(*^^^^^^^^^^^^^^^^^^^^^^^^^^^^^^^^^^^^^^ General Visualization ^^^^^^^^^^^^^^^^^^^^^^^^^^^^^^^^^^^^*)
	(*For Ready to Load Indicators*)
		(*Flash when tool should be loaded but load is not complete*)
		IF In_Auto AND Tool_At_Home AND NOT Welding_Complete AND All_Robots_Clear AND NOT All_Sensors_On.2
			THEN
				Ready_To_Load:= Pulse_500mS;
				(*Go solid when tool has been loaded properly*)
				(*Go solid when tool is ready to be unloaded*)
		ELSIF In_Auto AND All_Robots_Clear  AND ((Tool_At_Home AND NOT Welding_Complete AND All_Sensors_On.2 AND NOT Enable_Motion)
			OR (Tool_At_Unload.0 AND Welding_Complete AND (Sealing_Complete OR Sealer_Bypass) AND (Stud_Complete OR Stud_Bypass) AND TurntableA_At_Robot AND NOT All_Sensors_Off))
			THEN
				Ready_To_Load:= TRUE;
		ELSE
				Ready_To_Load:= FALSE;
		END_IF;
	(*For Red Stack Light Indicators*)
		Red_Lamp_Req:= PPFaults<>0 OR CLFaulted.0 OR CLFaulted.4 OR (NOT Sealer_Bypass AND MAIN.SL01.Disp1_Volume_NotOK AND (MAIN.R1.Task_ID_Ack=Seal_Fix16)) OR Load_Seq01.Faulted;


	(*Status Banners*)
		(*1 - Check Parts On Sub Check*)
		IF In_Auto AND NOT In_Manual AND NOT Cycle_Complete AND Tool_At_Load.0
			AND NOT Start_Load_Robots1 AND NOT Start_Load_Robots2 AND NOT Start_Seal_Robots AND NOT Start_Stud_Robots AND NOT Start_TurntableA
			AND NOT Start_TurntableB AND NOT Start_Weld_Robots AND NOT Start_Unload_Robots1 AND NOT Start_Unload_Robots2
			THEN
				IF NOT Dry_Cycle AND NOT All_Sensors_On.0
					THEN Status:= 1;
				ELSIF Dry_Cycle AND NOT Load_Complete1
					THEN Status:=1;
				END_IF;
		END_IF;
		(*2 - Sub Check OK*)
		IF In_Auto AND NOT In_Manual AND NOT Cycle_Complete AND Tool_At_Load.1
			AND NOT Start_Load_Robots1 AND NOT Start_Load_Robots2 AND NOT Start_Seal_Robots AND NOT Start_Stud_Robots AND NOT Start_TurntableA
			AND NOT Start_TurntableB AND NOT Start_Weld_Robots AND NOT Start_Unload_Robots1 AND NOT Start_Unload_Robots2
			THEN
				IF NOT Dry_Cycle AND NOT All_Sensors_On.1
					THEN Status:= 2;
				ELSIF Dry_Cycle AND NOT Load_Complete2
					THEN Status:=2;
				END_IF;
		END_IF;
		(*3 - Load Main Part*)
		IF In_Auto AND NOT In_Manual AND NOT Cycle_Complete AND Tool_At_Home
			AND NOT Start_Load_Robots1 AND NOT Start_Load_Robots2 AND NOT Start_Seal_Robots AND NOT Start_Stud_Robots AND NOT Start_TurntableA
			AND NOT Start_TurntableB AND NOT Start_Weld_Robots AND NOT Start_Unload_Robots1 AND NOT Start_Unload_Robots2
			THEN
				IF NOT Dry_Cycle AND NOT All_Sensors_On.2
					THEN Status:= 3;
				ELSIF Dry_Cycle AND NOT Load_Complete
					THEN Status:=3;
				END_IF;
		END_IF;
		(*10 - Load Parts Onto Tool*)
		IF In_Auto AND NOT In_Manual AND NOT Cycle_Complete AND Tool_At_Load.0
			AND NOT Start_Load_Robots1 AND NOT Start_Load_Robots2 AND NOT Start_Seal_Robots AND NOT Start_Stud_Robots AND NOT Start_TurntableA
			AND NOT Start_TurntableB AND NOT Start_Weld_Robots AND NOT Start_Unload_Robots1 AND NOT Start_Unload_Robots2
			THEN
				IF NOT Dry_Cycle AND NOT All_Sensors_On.2
					THEN Status:= 10;
				ELSIF Dry_Cycle AND NOT Load_Complete
					THEN Status:=10;
				END_IF;
		END_IF;
		(*11 - Robot(s) Loading*)
		IF ((Start_Load_Robots1 OR  Load_Robots_WorkingOK1) OR (Start_Load_Robots2 OR  Load_Robots_WorkingOK2)) AND In_Auto AND NOT In_Manual
			AND NOT Start_Seal_Robots AND NOT Start_Stud_Robots AND NOT Start_TurntableA
			AND NOT Start_TurntableB AND NOT Start_Weld_Robots AND NOT Start_Unload_Robots1 AND NOT Start_Unload_Robots2
			THEN Status:= 11;
		END_IF;
		(*12 - Parts Loaded OK*)
		IF In_Auto AND NOT In_Manual AND NOT Cycle_Complete
			AND NOT Start_Load_Robots1 AND NOT Start_Load_Robots2 AND NOT Start_Seal_Robots AND NOT Start_Stud_Robots AND NOT Start_TurntableA
			 AND NOT Start_TurntableB AND NOT Start_Weld_Robots AND NOT Start_Unload_Robots1 AND NOT Start_Unload_Robots2
			THEN
				IF (All_Sensors_On.2 AND Tool_At_Load.0) AND NOT Dry_Cycle
					THEN Status:= 12;
				ELSIF Load_Complete
					THEN Status:= 12;
				END_IF;
		END_IF;
		(*19 - Robot(s) Stud*)
		IF (Start_Stud_Robots OR Stud_Robots_WorkingOK) AND In_Auto AND NOT In_Manual
			AND NOT Start_Load_Robots1 AND NOT Start_Load_Robots2 AND NOT Start_Weld_Robots AND NOT Start_Seal_Robots AND NOT Start_TurntableA
			 AND NOT Start_TurntableB AND NOT Start_Unload_Robots1 AND NOT Start_Unload_Robots2
			THEN Status:= 19;
		END_IF;
		(*20 - Robot(s) Sealing*)
		IF (Start_Seal_Robots OR Seal_Robots_WorkingOK) AND In_Auto AND NOT In_Manual
			AND NOT Start_Load_Robots1 AND NOT Start_Load_Robots2 AND NOT Start_Weld_Robots AND NOT Start_Stud_Robots AND NOT Start_TurntableA
			 AND NOT Start_TurntableB AND NOT Start_Unload_Robots1 AND NOT Start_Unload_Robots2
			THEN Status:= 20;
		END_IF;
		(*21 - Robot(s) Welding*)
		IF (Start_Weld_Robots OR Weld_Robots_WorkingOK) AND In_Auto AND NOT In_Manual
			AND NOT Start_Load_Robots1 AND NOT Start_Load_Robots2 AND NOT Start_Seal_Robots AND NOT Start_Stud_Robots AND NOT Start_TurntableA
			 AND NOT Start_TurntableB AND NOT Start_Unload_Robots1 AND NOT Start_Unload_Robots2
			THEN Status:= 21;
		END_IF;
		(*22 - Welding Complete / Ready for Unload*)
		IF In_Auto AND NOT In_Manual AND NOT Cycle_Complete AND Welding_Complete
			AND NOT Start_Load_Robots1 AND NOT Start_Load_Robots2 AND NOT Start_Seal_Robots AND NOT Start_Stud_Robots AND NOT Start_TurntableA
			AND NOT Start_TurntableB AND NOT Start_Weld_Robots AND NOT Start_Unload_Robots1 AND NOT Start_Unload_Robots2
			THEN Status:= 22;
		END_IF;
		(*26 - Ready for Rotate*)
		IF (Start_TurntableA OR Start_TurntableB) AND In_Auto AND NOT In_Manual
			AND NOT Start_Load_Robots1 AND NOT Start_Load_Robots2 AND NOT Start_Seal_Robots AND NOT Start_Stud_Robots
			AND NOT Start_Weld_Robots AND NOT Start_Unload_Robots1 AND NOT Start_Unload_Robots2
			THEN Status := 26;
		END_IF;
		(*31 - Robot(s) Unloading*)
		IF (Start_Unload_Robots1 OR Unload_Robots_WorkingOK1 OR Start_Unload_Robots2 OR Unload_Robots_WorkingOK2) AND In_Auto AND NOT In_Manual
			AND NOT Start_Load_Robots1 AND NOT Start_Load_Robots2 AND NOT Start_Seal_Robots AND NOT Start_Stud_Robots AND NOT Start_TurntableA
			AND NOT Start_TurntableB AND NOT Start_Weld_Robots
			THEN Status:= 31;
		END_IF;
		(*32 - Unload Complete*)
		IF In_Auto AND NOT In_Manual AND NOT Cycle_Complete AND Unload_Complete
			AND NOT Start_Load_Robots1 AND NOT Start_Load_Robots2 AND NOT Start_Seal_Robots AND NOT Start_Stud_Robots AND NOT Start_TurntableA
			AND NOT Start_TurntableB AND NOT Start_Weld_Robots AND NOT Start_Unload_Robots1 AND NOT Start_Unload_Robots2
			THEN Status:= 32;
		END_IF;
		(*42 - Cycle Complete*)
		IF In_Auto AND NOT In_Manual AND Cycle_Complete AND All_Sensors_Off
			THEN Status:= 42;
		END_IF;
		(*50 - In Manual*)
		IF In_Manual
			THEN Status:= 50;
		END_IF;
		(*51 - Clamp Fault*)
		IF (CLFaults1>0 OR CLFaults2>0 OR CLFaults3>0 OR CLFaults4>0) AND In_Auto AND NOT In_Manual
			THEN Status:= 51;
		END_IF;
		(*52 - Part Present Sensor Fault*)
		IF PPFaults>0 AND In_Auto AND NOT In_Manual
			THEN Status:= 52;
		END_IF;
		(*53 - Nut Checks Failed Call QA*)
		IF QAChecks_Failed AND In_Auto AND NOT In_Manual
			THEN Status:= 53;
		END_IF;
		(*54 - Sealer Failed Call QA*)
		IF NOT Sealer_Bypass AND (MAIN.SL01.Disp1_Volume_NotOK AND (MAIN.R1.Task_ID_Ack=Seal_Fix16)) AND In_Auto AND NOT In_Manual
			THEN Status:= 54;
		END_IF;
		(*55 - Load Sequence Fault Call QA*)
		IF Load_Seq01.Faulted AND In_Auto AND NOT In_Manual
			THEN Status:= 55;
		END_IF;



(*$$$$$$$$$$$$$$$$$$$$$$$$$$$$$$$$$$$$$$$$$$$$$$$$$$$ Faults $$$$$$$$$$$$$$$$$$$$$$$$$$$$$$$$$$$$$$$$$$$$$$$$$$$$$$$*)

	(*Clamp/Cylider Faults Group 1*)
		IF CLFaults1>0
			THEN CLFaulted.1:=TRUE;
		ELSE
			CLFaulted.1:=FALSE;
		END_IF;
	(*Clamp/Cylider Faults Group 2*)
		IF CLFaults2>0
			THEN CLFaulted.2:=TRUE;
		ELSE
			CLFaulted.2:=FALSE;
		END_IF;
	(*Clamp/Cylider Faults Group 3*)
		IF CLFaults3>0
			THEN CLFaulted.3:=TRUE;
		ELSE
			CLFaulted.3:=FALSE;
		END_IF;
	(*Clamp/Cylinder Faults Group 4 - Reserved Flag for QA Check Motion Faults*)
		IF CLFaults4>0
			THEN CLFaulted.4:=TRUE;
		ELSE
			CLFaulted.4:=FALSE;
		END_IF;
	(*Bit 0 is designated as ANY Clamp Group Faulted*)
	IF CLFaulted.1 OR CLFaulted.2 OR CLFaulted.3
		THEN CLFaulted.0:= TRUE;
	ELSE CLFaulted.0 := FALSE;
	END_IF;

	(*Part Present Sensor Faults*)
		IF (PPFaults>0) OR (PPFaults1>0) OR (PPFaults2>0)
			THEN PPFaulted.0:=TRUE;
		ELSE
			PPFaulted.0:=FALSE;
		END_IF;
























(*end*)
END_ACTION

ACTION Task_Fix_Model_IDs:


	(*Develop Task IDs - See Global Variable, "TaskID_Record"*)

	IF (Start_Load_Robots1 OR Start_Load_Robots2) AND Enable_Motion
		THEN Task_ID:= Dropoff_Fix112;
	ELSIF Start_Seal_Robots AND Enable_Motion
		THEN Task_ID:= Seal_Fix112;
	ELSIF Start_Stud_Robots AND Enable_Motion
		THEN Task_ID:= Stud_Fix112;
	ELSIF Start_Weld_Robots AND Enable_Motion
		THEN Task_ID:= Weld_Fix112;
	ELSIF Start_TurnTableA AND Enable_Motion
		THEN Task_ID:= Sweep_Fix112;
	ELSIF (Start_Unload_Robots1 OR Start_Unload_Robots2) AND Enable_Motion
		THEN Task_ID:= Pickup_Fix112;
	ELSE Task_ID:= 0;
	END_IF;

	(*Develop Fixture ID*)
	Fix_ID:= N00.ID;					(*In Future Map Beckhoff Dip Switch Data From IP67 Block to Here*)

	(*Develop Model ID*)
	Model_ID:= Discrete_In.ModelData;
END_ACTION

ACTION Tool_States:


(*+++++++++++THIS AREA IS CUSTOM PER INSTALLATION AND WILL HAVE TO BE MODIFIED PER +++++++++++++*)
(*+++++++++++THIS AREA IS CUSTOM PER INSTALLATION AND WILL HAVE TO BE MODIFIED PER +++++++++++++*)

	Tool_At_HOME:= Clamp1RETD AND Clamp2RETD AND Clamp3RETD AND Clamp4RETD
				AND Clamp5RETD AND Clamp6RETD AND Clamp7RETD AND Clamp8RETD
				AND Clamp9RETD AND Clamp10RETD AND Clamp11RETD AND Clamp12RETD
				AND Clamp13RETD AND Clamp14RETD AND Clamp15RETD AND Clamp16RETD
				AND Clamp17RETD AND Clamp18RETD AND Clamp19RETD AND Clamp20RETD
				AND Clamp21RETD AND Clamp22RETD AND Clamp23RETD AND Clamp24RETD
				AND Pin1ADVD AND Pin2ADVD AND Pin3ADVD AND Pin4ADVD AND Pin5ADVD AND Pin6ADVD AND Pin7ADVD
				AND Pin8ADVD AND Pin9ADVD AND Pin10ADVD AND Pin11ADVD AND Pin12ADVD AND Pin13ADVD AND Pin14ADVD
				AND Slide1RETD AND Slide2RETD AND Slide3RETD AND Slide4RETD AND Slide5RETD AND Slide6RETD
				AND Swing1ADVD AND Swing2ADVD AND Swing3ADVD AND Swing4ADVD AND Swing5ADVD AND Swing6ADVD;


	Tool_At_Load.0:=Clamp1RETD AND Clamp2RETD AND Clamp3RETD AND Clamp4RETD
				AND Clamp5RETD AND Clamp6RETD AND Clamp7RETD AND Clamp8RETD
				AND Clamp9RETD AND Clamp10RETD AND Clamp11RETD AND Clamp12RETD
				AND Clamp13RETD AND Clamp14RETD AND Clamp15RETD AND Clamp16RETD
				AND Clamp17RETD AND Clamp18RETD AND Clamp19RETD AND Clamp20RETD
				AND Clamp21RETD AND Clamp22RETD AND Clamp23RETD AND Clamp24RETD
				AND Pin1ADVD AND Pin2ADVD AND Pin3ADVD AND Pin4ADVD AND Pin5ADVD AND Pin6ADVD AND Pin7ADVD
				AND Pin8ADVD AND Pin9ADVD AND Pin10ADVD AND Pin11ADVD AND Pin12ADVD AND Pin13ADVD AND Pin14ADVD
				AND Slide1RETD AND Slide2RETD AND Slide3RETD AND Slide4RETD AND Slide5RETD AND Slide6RETD
				AND Swing1ADVD AND Swing2ADVD AND Swing3ADVD AND Swing4ADVD AND Swing5ADVD AND Swing6ADVD;
	Tool_At_Load.1:=FALSE;
	Tool_At_Load.2:= FALSE;
	Tool_At_Load.3:= FALSE;
	Tool_At_Load.4:= FALSE;


	Tool_At_Seal.0:= Clamp1ADVD AND Clamp2ADVD AND Clamp3ADVD AND Clamp4ADVD
				AND Clamp5ADVD AND Clamp6ADVD AND Clamp7ADVD AND Clamp8ADVD
				AND Clamp9ADVD AND Clamp10ADVD AND Clamp11ADVD AND Clamp12ADVD
				AND Clamp13ADVD AND Clamp14ADVD AND Clamp15ADVD AND Clamp16ADVD
				AND Clamp17ADVD AND Clamp18ADVD AND Clamp19ADVD AND Clamp20ADVD
				AND Clamp21ADVD AND Clamp22ADVD AND Clamp23ADVD AND Clamp24ADVD
				AND Pin1ADVD AND Pin2ADVD AND Pin3ADVD AND Pin4ADVD AND Pin5ADVD AND Pin6ADVD AND Pin7ADVD
				AND Pin8ADVD AND Pin9ADVD AND Pin10ADVD AND Pin11ADVD AND Pin12ADVD AND Pin13ADVD AND Pin14ADVD
				AND Slide1RETD AND Slide2RETD AND Slide3RETD AND Slide4RETD AND Slide5RETD AND Slide6RETD
				AND Swing1ADVD AND Swing2ADVD AND Swing3ADVD AND Swing4ADVD AND Swing5ADVD AND Swing6ADVD;
	Tool_At_Seal.1:= FALSE;
	Tool_At_Seal.2:= FALSE;
	Tool_At_Seal.3:= FALSE;
	Tool_At_Seal.4:= FALSE;


	Tool_At_Stud.0:= Clamp1ADVD AND Clamp2ADVD AND Clamp3ADVD AND Clamp4ADVD
				AND Clamp5ADVD AND Clamp6ADVD AND Clamp7ADVD AND Clamp8ADVD
				AND Clamp9ADVD AND Clamp10ADVD AND Clamp11ADVD AND Clamp12ADVD
				AND Clamp13ADVD AND Clamp14ADVD AND Clamp15ADVD AND Clamp16ADVD
				AND Clamp17ADVD AND Clamp18ADVD AND Clamp19ADVD AND Clamp20ADVD
				AND Clamp21ADVD AND Clamp22ADVD AND Clamp23ADVD AND Clamp24ADVD
				AND Pin1ADVD AND Pin2ADVD AND Pin3ADVD AND Pin4ADVD AND Pin5ADVD AND Pin6ADVD AND Pin7ADVD
				AND Pin8ADVD AND Pin9ADVD AND Pin10ADVD AND Pin11ADVD AND Pin12ADVD AND Pin13ADVD AND Pin14ADVD
				AND Slide1RETD AND Slide2RETD AND Slide3RETD AND Slide4RETD AND Slide5RETD AND Slide6RETD
				AND Swing1ADVD AND Swing2ADVD AND Swing3ADVD AND Swing4ADVD AND Swing5ADVD AND Swing6ADVD;
	Tool_At_Stud.1:= FALSE;
	Tool_At_Stud.2:= FALSE;
	Tool_At_Stud.3:= FALSE;
	Tool_At_Stud.4:= FALSE;


	Tool_At_Rotate.0:= Clamp1ADVD AND Clamp2ADVD AND Clamp3ADVD AND Clamp4ADVD
				AND Clamp5ADVD AND Clamp6ADVD AND Clamp7ADVD AND Clamp8ADVD
				AND Clamp9ADVD AND Clamp10ADVD AND Clamp11ADVD AND Clamp12ADVD
				AND Clamp13ADVD AND Clamp14ADVD AND Clamp15ADVD AND Clamp16ADVD
				AND Clamp17ADVD AND Clamp18ADVD AND Clamp19ADVD AND Clamp20ADVD
				AND Clamp21ADVD AND Clamp22ADVD AND Clamp23ADVD AND Clamp24ADVD
				AND Pin1ADVD AND Pin2ADVD AND Pin3ADVD AND Pin4ADVD AND Pin5ADVD AND Pin6ADVD AND Pin7ADVD
				AND Pin8ADVD AND Pin9ADVD AND Pin10ADVD AND Pin11ADVD AND Pin12ADVD AND Pin13ADVD AND Pin14ADVD
				AND Slide1RETD AND Slide2RETD AND Slide3RETD AND Slide4RETD AND Slide5RETD AND Slide6RETD
				AND Swing1ADVD AND Swing2ADVD AND Swing3ADVD AND Swing4ADVD AND Swing5ADVD AND Swing6ADVD;
	Tool_At_Rotate.1:= FALSE;
	Tool_At_Rotate.2:= FALSE;
	Tool_At_Rotate.3:= FALSE;
	Tool_At_Rotate.4:= FALSE;


	Tool_At_Weld.0:= Clamp1ADVD AND Clamp2ADVD AND Clamp3ADVD AND Clamp4ADVD
				AND Clamp5ADVD AND Clamp6ADVD AND Clamp7ADVD AND Clamp8ADVD
				AND Clamp9ADVD AND Clamp10ADVD AND Clamp11ADVD AND Clamp12ADVD
				AND Clamp13ADVD AND Clamp14ADVD AND Clamp15ADVD AND Clamp16ADVD
				AND Clamp17ADVD AND Clamp18ADVD AND Clamp19ADVD AND Clamp20ADVD
				AND Clamp21ADVD AND Clamp22ADVD AND Clamp23ADVD AND Clamp24ADVD
				AND Pin1ADVD AND Pin2ADVD AND Pin3ADVD AND Pin4ADVD AND Pin5ADVD AND Pin6ADVD AND Pin7ADVD
				AND Pin8ADVD AND Pin9ADVD AND Pin10ADVD AND Pin11ADVD AND Pin12ADVD AND Pin13ADVD AND Pin14ADVD
				AND Slide1RETD AND Slide2RETD AND Slide3RETD AND Slide4RETD AND Slide5RETD AND Slide6RETD
				AND Swing1ADVD AND Swing2ADVD AND Swing3ADVD AND Swing4ADVD AND Swing5ADVD AND Swing6ADVD;
	Tool_At_Weld.1:= FALSE;
	Tool_At_Weld.2:= FALSE;
	Tool_At_Weld.3:= FALSE;
	Tool_At_Weld.4:= FALSE;


	Tool_At_Unload.0:=Clamp1RETD AND Clamp2RETD AND Clamp3RETD AND Clamp4RETD
				AND Clamp5RETD AND Clamp6RETD AND Clamp7RETD AND Clamp8RETD
				AND Clamp9RETD AND Clamp10RETD AND Clamp11RETD AND Clamp12RETD
				AND Clamp13RETD AND Clamp14RETD AND Clamp15RETD AND Clamp16RETD
				AND Clamp17RETD AND Clamp18RETD AND Clamp19RETD AND Clamp20RETD
				AND Clamp21RETD AND Clamp22RETD AND Clamp23RETD AND Clamp24RETD
				AND Pin1RETD AND Pin2RETD AND Pin3RETD AND Pin4RETD AND Pin5RETD AND Pin6RETD AND Pin7RETD
				AND Pin8RETD AND Pin9RETD AND Pin10RETD AND Pin11RETD AND Pin12RETD AND Pin13RETD AND Pin14RETD
				AND Slide1ADVD AND Slide2ADVD AND Slide3ADVD AND Slide4ADVD AND Slide5ADVD AND Slide6ADVD
				AND Swing1RETD AND Swing2RETD AND Swing3RETD AND Swing4RETD AND Swing5RETD AND Swing6RETD;
	Tool_At_Unload.1:=FALSE;
	Tool_At_Unload.2:= FALSE;
	Tool_At_Unload.3:= FALSE;
	Tool_At_Unload.4:= FALSE;







































(*end*)
END_ACTION

ACTION Tool_VBSeq_Repos:
(*+++++++++++THIS AREA IS CUSTOM PER INSTALLATION AND WILL HAVE TO BE MODIFIED PER +++++++++++++*)
(*+++++++++++THIS AREA IS CUSTOM PER INSTALLATION AND WILL HAVE TO BE MODIFIED PER +++++++++++++*)


(*!!!!!!!!!!!!!!!!!!!!!!!!!!!!!!!!!!!!!!!!!! Tool Motion Control !!!!!!!!!!!!!!!!!!!!!!!!!!!!!!!*)

(*----------------------------------------- Camp / Unclamp Steps -------------------------------*)

(*$$$$$$$$$$$$$$$$$$$$$$$$$$$$$$$$$$ Develop Clamp and Unclamp Interlocks $$$$$$$$$$$$$$$$$$$$$$*)
(* Note: This is one method to create valve bank commands for clamp and unclamp sequencing
you are welcome to use the direct method as well*)

	(*Start Clamp Sequence*)
	(*First Stage Clamping*)
	Clamp_Step.0:= Auto_Run AND NOT Welding_Complete AND FALSE;
	(*Second Stage Clamping*)
	Clamp_Step.1:=  Clamp_Step.0 AND FALSE;
	(*Third Stage Clamping*)
	Clamp_Step.2:= Clamp_Step.1 AND FALSE;
	(*Forth Stage Clamping*)
	Clamp_Step.3:= Clamp_Step.2 AND FALSE;


	(*Start Unlcamp Sequence*)
	(*First Stage Unclamping*)
	Unclamp_Step.0:= Welding_Complete AND FALSE;
	(*Second Stage Unclamping*)
	Unclamp_Step.1:= Unclamp_Step.0 AND FALSE;
	(*Third Stage Unclamping*)
	Unclamp_Step.2:= Unclamp_Step.1 AND FALSE;
	(*Fourth Stage Unclamping*)
	Unclamp_Step.3:= Unclamp_Step.2 AND FALSE;



(*------------------------------------------- Repositions --------------------------------------*)

	(*Reposition Request#1*)
	IF FALSE
		THEN
			Repo_Reqs.0:= TRUE;
	END_IF;

	(*Reposition Request#2*)
	IF FALSE
		THEN
			Repo_Reqs.1:= TRUE;
	END_IF;

	(*Reposition Request#3*)
	IF FALSE
		THEN
			Repo_Reqs.2:= TRUE;
	END_IF;

	(*Reposition Request#4*)
	IF FALSE
		THEN
			Repo_Reqs.3:= TRUE;
	END_IF;

	(*Reposition Request#5*)
	IF FALSE
		THEN
			Repo_Reqs.4:= TRUE;
	END_IF;

	(*Reposition Request#6*)
	IF FALSE
		THEN
			Repo_Reqs.5:= TRUE;
	END_IF;

	(*Reposition Request#7*)
	IF FALSE
		THEN
			Repo_Reqs.6:= TRUE;
	END_IF;

	(*Reposition Request#8*)
	IF FALSE
		THEN
			Repo_Reqs.7:= TRUE;
	END_IF;

	(*Reset All Reposition Acks At the End Of Cycle*)
	IF Cycle_Complete
		THEN
			Repo_Reqs:= 0;
	END_IF;

(*------------------------- Reposition Acks ---------------------*)
	Repo_Ack.0:= Repo_Reqs.0 AND FALSE;
	Repo_Ack.1:= Repo_Reqs.1 AND FALSE;
	Repo_Ack.2:= Repo_Reqs.2 AND FALSE;
	Repo_Ack.3:= Repo_Reqs.3 AND FALSE;
	Repo_Ack.4:= Repo_Reqs.4 AND FALSE;
	Repo_Ack.5:= Repo_Reqs.5 AND FALSE;
	Repo_Ack.6:= Repo_Reqs.6 AND FALSE;
	Repo_Ack.7:= Repo_Reqs.7 AND FALSE;
END_ACTION

ACTION ValveBank1:


(*+++++++++++THIS AREA IS CUSTOM PER INSTALLATION AND WILL HAVE TO BE MODIFIED PER +++++++++++++*)
(*+++++++++++THIS AREA IS CUSTOM PER INSTALLATION AND WILL HAVE TO BE MODIFIED PER +++++++++++++*)
(*+++++++++++THIS AREA IS CUSTOM PER INSTALLATION AND WILL HAVE TO BE MODIFIED PER +++++++++++++*)

(*+++++++++++VALVE BANK 1 +++++++++++++*)
(*+++++++++++VALVE BANK 1 +++++++++++++*)
(*+++++++++++VALVE BANK 1 +++++++++++++*)


	(*Valve 1, A+B*)
	(*spare*)
		Valve1FB
			(
			Enable_Motion:= Enable_Motion ,
			Enable_Latch:= TRUE,					(*Enabling Runs Valve as detent type (maintained solenoids*)
			Enable_SideA_PreCharge:= FALSE,		(*Enabling Turns Side A PreCharge Active, reset when Side B is energized in Auto*)
			Enable_SideB_PreCharge:= FALSE,		(*Enabling Turns Side B PreCharge Active, reset when Side A is energized in Auto*)
			PreCharge_Time:= T#0.1S,
			Enable_Auto_Commands:= In_Auto,
			Enable_Manual_Commands:= In_Manual AND All_Robots_Clear,
			In_Manual_SideA_Command:= Discrete_In.ManReqs.0,
			In_Manual_SideB_Command:= (Discrete_In.ManReqs.1 OR Discrete_In.Go_Home),
			SideA_Indicator:= (Clamp1ADVD AND Clamp2ADVD AND Clamp3ADVD AND Clamp4ADVD),
			SideB_Indicator:= (Clamp1RETD AND Clamp2RETD AND Clamp3RETD AND Clamp4RETD) OR Manual_Ind_HomePrompt,
			TurnOn_SideA_SOL=> N100.Q.0,
			TurnOn_SideB_SOL=> N100.Q.1,
			TurnOn_SideA_Indicator=> Manual_Indicators1.0,
			TurnOn_SideB_Indicator=> Manual_Indicators1.1
			 );
		Valve1FB.In_Auto_SideA_Command:= FALSE;
		Valve1FB.In_Auto_SideB_Command:= FALSE;


	(*Valve 2, A+B*)
	(*spare*)
		Valve2FB
			(
			Enable_Motion:= Enable_Motion ,
			Enable_Latch:= TRUE,					(*Enabling Runs Valve as detent type (maintained solenoids*)
			Enable_SideA_PreCharge:= FALSE,		(*Enabling Turns Side A PreCharge Active, reset when Side B is energized in Auto*)
			Enable_SideB_PreCharge:= FALSE,		(*Enabling Turns Side B PreCharge Active, reset when Side A is energized in Auto*)
			PreCharge_Time:= T#0.10S,
			Enable_Auto_Commands:= In_Auto,
			Enable_Manual_Commands:= In_Manual AND All_Robots_Clear,
			In_Manual_SideA_Command:= Discrete_In.ManReqs.2,
			In_Manual_SideB_Command:= Discrete_In.ManReqs.3,
			SideA_Indicator:= FALSE,
			SideB_Indicator:= FALSE,
			TurnOn_SideA_SOL=> N100.Q.2,
			TurnOn_SideB_SOL=> N100.Q.3,
			TurnOn_SideA_Indicator=> Manual_Indicators1.2,
			TurnOn_SideB_Indicator=> Manual_Indicators1.3
			 );
		Valve2FB.In_Auto_SideA_Command:= FALSE;
		Valve2FB.In_Auto_SideB_Command:= FALSE;


	(*Valve 3, A+B*)
	(*spare*)
		Valve3FB
			(
			Enable_Motion:= Enable_Motion ,
			Enable_Latch:= TRUE,					(*Enabling Runs Valve as detent type (maintained solenoids*)
			Enable_SideA_PreCharge:= FALSE,		(*Enabling Turns Side A PreCharge Active, reset when Side B is energized in Auto*)
			Enable_SideB_PreCharge:= FALSE,		(*Enabling Turns Side B PreCharge Active, reset when Side A is energized in Auto*)
			PreCharge_Time:= T#0.10S,
			Enable_Auto_Commands:= In_Auto,
			Enable_Manual_Commands:= In_Manual AND All_Robots_Clear,
			In_Manual_SideA_Command:= Discrete_In.ManReqs.4,
			In_Manual_SideB_Command:= Discrete_In.ManReqs.5,
			SideA_Indicator:= FALSE,
			SideB_Indicator:= FALSE,
			TurnOn_SideA_SOL=> N100.Q.4,
			TurnOn_SideB_SOL=> N100.Q.5,
			TurnOn_SideA_Indicator=> Manual_Indicators1.4,
			TurnOn_SideB_Indicator=> Manual_Indicators1.5
			 );
		Valve3FB.In_Auto_SideA_Command:= FALSE;
		Valve3FB.In_Auto_SideB_Command:= FALSE;


	(*Valve 4, A+B*)
	(*spare*)
		Valve4FB
			(
			Enable_Motion:= Enable_Motion ,
			Enable_Latch:= TRUE,					(*Enabling Runs Valve as detent type (maintained solenoids*)
			Enable_SideA_PreCharge:= FALSE,		(*Enabling Turns Side A PreCharge Active, reset when Side B is energized in Auto*)
			Enable_SideB_PreCharge:= FALSE,		(*Enabling Turns Side B PreCharge Active, reset when Side A is energized in Auto*)
			PreCharge_Time:= T#0.10S,
			Enable_Auto_Commands:= In_Auto,
			Enable_Manual_Commands:= In_Manual AND All_Robots_Clear,
			In_Manual_SideA_Command:= Discrete_In.ManReqs.6,
			In_Manual_SideB_Command:= Discrete_In.ManReqs.7,
			SideA_Indicator:= FALSE,
			SideB_Indicator:= FALSE,
			TurnOn_SideA_SOL=> N100.Q.6,
			TurnOn_SideB_SOL=> N100.Q.7,
			TurnOn_SideA_Indicator=> Manual_Indicators1.6,
			TurnOn_SideB_Indicator=> Manual_Indicators1.7
			 );
		Valve4FB.In_Auto_SideA_Command:= FALSE;
		Valve4FB.In_Auto_SideB_Command:= FALSE;


	(*Valve 5, A+B*)
	(*spare*)
		Valve5FB
			(
			Enable_Motion:= Enable_Motion ,
			Enable_Latch:= TRUE,					(*Enabling Runs Valve as detent type (maintained solenoids*)
			Enable_SideA_PreCharge:= FALSE,		(*Enabling Turns Side A PreCharge Active, reset when Side B is energized in Auto*)
			Enable_SideB_PreCharge:= FALSE,		(*Enabling Turns Side B PreCharge Active, reset when Side A is energized in Auto*)
			PreCharge_Time:= T#0.10S,
			Enable_Auto_Commands:= In_Auto,
			Enable_Manual_Commands:= In_Manual AND All_Robots_Clear,
			In_Manual_SideA_Command:= Discrete_In.ManReqs.8,
			In_Manual_SideB_Command:= Discrete_In.ManReqs.9,
			SideA_Indicator:= FALSE,
			SideB_Indicator:= FALSE,
			TurnOn_SideA_SOL=> N100.Q.8,
			TurnOn_SideB_SOL=> N100.Q.9,
			TurnOn_SideA_Indicator=> Manual_Indicators1.8,
			TurnOn_SideB_Indicator=> Manual_Indicators1.9
			 );
		Valve5FB.In_Auto_SideA_Command:= FALSE;
		Valve5FB.In_Auto_SideB_Command:= FALSE;


	(*Valve 6, A+B*)
	(*spare*)
		Valve6FB
			(
			Enable_Motion:= Enable_Motion ,
			Enable_Latch:= TRUE,					(*Enabling Runs Valve as detent type (maintained solenoids*)
			Enable_SideA_PreCharge:= FALSE,		(*Enabling Turns Side A PreCharge Active, reset when Side B is energized in Auto*)
			Enable_SideB_PreCharge:= FALSE,		(*Enabling Turns Side B PreCharge Active, reset when Side A is energized in Auto*)
			PreCharge_Time:= T#0.10S,
			Enable_Auto_Commands:= In_Auto,
			Enable_Manual_Commands:= In_Manual AND All_Robots_Clear,
			In_Manual_SideA_Command:= Discrete_In.ManReqs.10,
			In_Manual_SideB_Command:= Discrete_In.ManReqs.11,
			SideA_Indicator:= FALSE,
			SideB_Indicator:= FALSE,
			TurnOn_SideA_SOL=> N100.Q.10,
			TurnOn_SideB_SOL=> N100.Q.11,
			TurnOn_SideA_Indicator=> Manual_Indicators1.10,
			TurnOn_SideB_Indicator=> Manual_Indicators1.11
			 );
		Valve6FB.In_Auto_SideA_Command:= FALSE;
		Valve6FB.In_Auto_SideB_Command:= FALSE;


	(*Valve 7, A+B*)
	(*spare*)
		Valve7FB
			(
			Enable_Motion:= Enable_Motion ,
			Enable_Latch:= TRUE,					(*Enabling Runs Valve as detent type (maintained solenoids*)
			Enable_SideA_PreCharge:= FALSE,		(*Enabling Turns Side A PreCharge Active, reset when Side B is energized in Auto*)
			Enable_SideB_PreCharge:= FALSE,		(*Enabling Turns Side B PreCharge Active, reset when Side A is energized in Auto*)
			PreCharge_Time:= T#0.10S,
			Enable_Auto_Commands:= In_Auto,
			Enable_Manual_Commands:= In_Manual AND All_Robots_Clear,
			In_Manual_SideA_Command:= Discrete_In.ManReqs.12,
			In_Manual_SideB_Command:= Discrete_In.ManReqs.13,
			SideA_Indicator:= FALSE,
			SideB_Indicator:= FALSE,
			TurnOn_SideA_SOL=> N100.Q.12,
			TurnOn_SideB_SOL=> N100.Q.13,
			TurnOn_SideA_Indicator=> Manual_Indicators1.12,
			TurnOn_SideB_Indicator=> Manual_Indicators1.13
			 );
		Valve7FB.In_Auto_SideA_Command:= FALSE;
		Valve7FB.In_Auto_SideB_Command:= FALSE;


	(*Valve 8, A+B*)
	(*spare*)
		Valve8FB
			(
			Enable_Motion:= Enable_Motion ,
			Enable_Latch:= TRUE,					(*Enabling Runs Valve as detent type (maintained solenoids*)
			Enable_SideA_PreCharge:= FALSE,		(*Enabling Turns Side A PreCharge Active, reset when Side B is energized in Auto*)
			Enable_SideB_PreCharge:= FALSE,		(*Enabling Turns Side B PreCharge Active, reset when Side A is energized in Auto*)
			PreCharge_Time:= T#0.10S,
			Enable_Auto_Commands:= In_Auto,
			Enable_Manual_Commands:= In_Manual AND All_Robots_Clear,
			In_Manual_SideA_Command:= Discrete_In.ManReqs.14,
			In_Manual_SideB_Command:= Discrete_In.ManReqs.15,
			SideA_Indicator:= FALSE,
			SideB_Indicator:= FALSE,
			TurnOn_SideA_SOL=> N100.Q.14,
			TurnOn_SideB_SOL=> N100.Q.15,
			TurnOn_SideA_Indicator=> Manual_Indicators1.14,
			TurnOn_SideB_Indicator=> Manual_Indicators1.15
			 );
		Valve8FB.In_Auto_SideA_Command:= FALSE;
		Valve8FB.In_Auto_SideB_Command:= FALSE;


	(*Valve 9, A+B*)
	(*spare*)
		Valve9FB
			(
			Enable_Motion:= Enable_Motion ,
			Enable_Latch:= TRUE,					(*Enabling Runs Valve as detent type (maintained solenoids*)
			Enable_SideA_PreCharge:= FALSE,		(*Enabling Turns Side A PreCharge Active, reset when Side B is energized in Auto*)
			Enable_SideB_PreCharge:= FALSE,		(*Enabling Turns Side B PreCharge Active, reset when Side A is energized in Auto*)
			PreCharge_Time:= T#0.10S,
			Enable_Auto_Commands:= In_Auto,
			Enable_Manual_Commands:= In_Manual AND All_Robots_Clear,
			In_Manual_SideA_Command:= Discrete_In.ManReqs.16,
			In_Manual_SideB_Command:= Discrete_In.ManReqs.17,
			SideA_Indicator:= FALSE,
			SideB_Indicator:= FALSE,
			TurnOn_SideA_SOL=> N100.Q.16,
			TurnOn_SideB_SOL=> N100.Q.17,
			TurnOn_SideA_Indicator=> Manual_Indicators1.16,
			TurnOn_SideB_Indicator=> Manual_Indicators1.17
			 );
		Valve9FB.In_Auto_SideA_Command:= FALSE;
		Valve9FB.In_Auto_SideB_Command:= FALSE;


	(*Valve 10, A+B*)
	(*spare*)
		Valve10FB
			(
			Enable_Motion:= Enable_Motion ,
			Enable_Latch:= TRUE,					(*Enabling Runs Valve as detent type (maintained solenoids*)
			Enable_SideA_PreCharge:= FALSE,		(*Enabling Turns Side A PreCharge Active, reset when Side B is energized in Auto*)
			Enable_SideB_PreCharge:= FALSE,		(*Enabling Turns Side B PreCharge Active, reset when Side A is energized in Auto*)
			PreCharge_Time:= T#0.10S,
			Enable_Auto_Commands:= In_Auto,
			Enable_Manual_Commands:= In_Manual AND All_Robots_Clear,
			In_Manual_SideA_Command:= Discrete_In.ManReqs.18,
			In_Manual_SideB_Command:= Discrete_In.ManReqs.19,
			SideA_Indicator:= FALSE,
			SideB_Indicator:= FALSE,
			TurnOn_SideA_SOL=> N100.Q.18,
			TurnOn_SideB_SOL=> N100.Q.19,
			TurnOn_SideA_Indicator=> Manual_Indicators1.18,
			TurnOn_SideB_Indicator=> Manual_Indicators1.19
			 );
		Valve10FB.In_Auto_SideA_Command:= FALSE;
		Valve10FB.In_Auto_SideB_Command:= FALSE;


	(*Valve 11, A+B*)
	(*spare*)
		Valve11FB
			(
			Enable_Motion:= Enable_Motion ,
			Enable_Latch:= TRUE,					(*Enabling Runs Valve as detent type (maintained solenoids*)
			Enable_SideA_PreCharge:= FALSE,		(*Enabling Turns Side A PreCharge Active, reset when Side B is energized in Auto*)
			Enable_SideB_PreCharge:= FALSE,		(*Enabling Turns Side B PreCharge Active, reset when Side A is energized in Auto*)
			PreCharge_Time:= T#0.10S,
			Enable_Auto_Commands:= In_Auto,
			Enable_Manual_Commands:= In_Manual AND All_Robots_Clear,
			In_Manual_SideA_Command:= Discrete_In.ManReqs.20,
			In_Manual_SideB_Command:= Discrete_In.ManReqs.21,
			SideA_Indicator:= FALSE,
			SideB_Indicator:= FALSE,
			TurnOn_SideA_SOL=> N100.Q.20,
			TurnOn_SideB_SOL=> N100.Q.21,
			TurnOn_SideA_Indicator=> Manual_Indicators1.20,
			TurnOn_SideB_Indicator=> Manual_Indicators1.21
			 );
		Valve11FB.In_Auto_SideA_Command:= FALSE;
		Valve11FB.In_Auto_SideB_Command:= FALSE;


	(*Valve 12, A+B*)
	(*spare*)
		Valve12FB
			(
			Enable_Motion:= Enable_Motion ,
			Enable_Latch:= TRUE,					(*Enabling Runs Valve as detent type (maintained solenoids*)
			Enable_SideA_PreCharge:= FALSE,		(*Enabling Turns Side A PreCharge Active, reset when Side B is energized in Auto*)
			Enable_SideB_PreCharge:= FALSE,		(*Enabling Turns Side B PreCharge Active, reset when Side A is energized in Auto*)
			PreCharge_Time:= T#0.10S,
			Enable_Auto_Commands:= In_Auto,
			Enable_Manual_Commands:= In_Manual AND All_Robots_Clear,
			In_Manual_SideA_Command:= Discrete_In.ManReqs.22,
			In_Manual_SideB_Command:= Discrete_In.ManReqs.23,
			SideA_Indicator:= FALSE,
			SideB_Indicator:= FALSE,
			TurnOn_SideA_SOL=> N100.Q.22,
			TurnOn_SideB_SOL=> N100.Q.23,
			TurnOn_SideA_Indicator=> Manual_Indicators1.22,
			TurnOn_SideB_Indicator=> Manual_Indicators1.23
			 );
		Valve12FB.In_Auto_SideA_Command:= FALSE;
		Valve12FB.In_Auto_SideB_Command:= FALSE;


	(*Valve 13, A+B*)
	(*spare*)
		Valve13FB
			(
			Enable_Motion:= Enable_Motion ,
			Enable_Latch:= TRUE,					(*Enabling Runs Valve as detent type (maintained solenoids*)
			Enable_SideA_PreCharge:= FALSE,		(*Enabling Turns Side A PreCharge Active, reset when Side B is energized in Auto*)
			Enable_SideB_PreCharge:= FALSE,		(*Enabling Turns Side B PreCharge Active, reset when Side A is energized in Auto*)
			PreCharge_Time:= T#0.10S,
			Enable_Auto_Commands:= In_Auto,
			Enable_Manual_Commands:= In_Manual AND All_Robots_Clear,
			In_Manual_SideA_Command:= Discrete_In.ManReqs.24,
			In_Manual_SideB_Command:= Discrete_In.ManReqs.25,
			SideA_Indicator:= FALSE,
			SideB_Indicator:= FALSE,
			TurnOn_SideA_SOL=> N100.Q.24,
			TurnOn_SideB_SOL=> N100.Q.25,
			TurnOn_SideA_Indicator=> Manual_Indicators1.24,
			TurnOn_SideB_Indicator=> Manual_Indicators1.25
			 );
		Valve13FB.In_Auto_SideA_Command:= FALSE;
		Valve13FB.In_Auto_SideB_Command:= FALSE;


	(*Valve 14, A+B*)
	(*spare*)
		Valve14FB
			(
			Enable_Motion:= Enable_Motion ,
			Enable_Latch:= TRUE,					(*Enabling Runs Valve as detent type (maintained solenoids*)
			Enable_SideA_PreCharge:= FALSE,		(*Enabling Turns Side A PreCharge Active, reset when Side B is energized in Auto*)
			Enable_SideB_PreCharge:= FALSE,		(*Enabling Turns Side B PreCharge Active, reset when Side A is energized in Auto*)
			PreCharge_Time:= T#0.10S,
			Enable_Auto_Commands:= In_Auto,
			Enable_Manual_Commands:= In_Manual AND All_Robots_Clear,
			In_Manual_SideA_Command:= Discrete_In.ManReqs.26,
			In_Manual_SideB_Command:= Discrete_In.ManReqs.27,
			SideA_Indicator:= FALSE,
			SideB_Indicator:= FALSE,
			TurnOn_SideA_SOL=> N100.Q.26,
			TurnOn_SideB_SOL=> N100.Q.27,
			TurnOn_SideA_Indicator=> Manual_Indicators1.26,
			TurnOn_SideB_Indicator=> Manual_Indicators1.27
			 );
		Valve14FB.In_Auto_SideA_Command:= FALSE;
		Valve14FB.In_Auto_SideB_Command:= FALSE;


	(*Valve 15, A+B*)
	(*spare*)
		Valve15FB
			(
			Enable_Motion:= Enable_Motion ,
			Enable_Latch:= TRUE,					(*Enabling Runs Valve as detent type (maintained solenoids*)
			Enable_SideA_PreCharge:= FALSE,		(*Enabling Turns Side A PreCharge Active, reset when Side B is energized in Auto*)
			Enable_SideB_PreCharge:= FALSE,		(*Enabling Turns Side B PreCharge Active, reset when Side A is energized in Auto*)
			PreCharge_Time:= T#0.10S,
			Enable_Auto_Commands:= In_Auto,
			Enable_Manual_Commands:= In_Manual AND All_Robots_Clear,
			In_Manual_SideA_Command:= Discrete_In.ManReqs.28,
			In_Manual_SideB_Command:= Discrete_In.ManReqs.29,
			SideA_Indicator:= FALSE,
			SideB_Indicator:= FALSE,
			TurnOn_SideA_SOL=> N100.Q.28,
			TurnOn_SideB_SOL=> N100.Q.29,
			TurnOn_SideA_Indicator=> Manual_Indicators1.28,
			TurnOn_SideB_Indicator=> Manual_Indicators1.29
			 );
		Valve15FB.In_Auto_SideA_Command:= FALSE;
		Valve15FB.In_Auto_SideB_Command:= FALSE;


	(*Valve 16, A+B*)
	(*spare*)
		Valve16FB
			(
			Enable_Motion:= Enable_Motion ,
			Enable_Latch:= TRUE,					(*Enabling Runs Valve as detent type (maintained solenoids*)
			Enable_SideA_PreCharge:= FALSE,		(*Enabling Turns Side A PreCharge Active, reset when Side B is energized in Auto*)
			Enable_SideB_PreCharge:= FALSE,		(*Enabling Turns Side B PreCharge Active, reset when Side A is energized in Auto*)
			PreCharge_Time:= T#0.10S,
			Enable_Auto_Commands:= In_Auto,
			Enable_Manual_Commands:= In_Manual AND All_Robots_Clear,
			In_Manual_SideA_Command:= Discrete_In.ManReqs.30,
			In_Manual_SideB_Command:= Discrete_In.ManReqs.31,
			SideA_Indicator:= FALSE,
			SideB_Indicator:= FALSE,
			TurnOn_SideA_SOL=> N100.Q.30,
			TurnOn_SideB_SOL=> N100.Q.31,
			TurnOn_SideA_Indicator=> Manual_Indicators1.30,
			TurnOn_SideB_Indicator=> Manual_Indicators1.31
			 );
		Valve16FB.In_Auto_SideA_Command:= FALSE;
		Valve16FB.In_Auto_SideB_Command:= FALSE;


























(*end*)
END_ACTION

ACTION ValveBank2:


(*+++++++++++THIS AREA IS CUSTOM PER INSTALLATION AND WILL HAVE TO BE MODIFIED PER +++++++++++++*)
(*+++++++++++THIS AREA IS CUSTOM PER INSTALLATION AND WILL HAVE TO BE MODIFIED PER +++++++++++++*)
(*+++++++++++THIS AREA IS CUSTOM PER INSTALLATION AND WILL HAVE TO BE MODIFIED PER +++++++++++++*)

(*+++++++++++VALVE BANK 2 +++++++++++++*)
(*+++++++++++VALVE BANK 2 +++++++++++++*)
(*+++++++++++VALVE BANK 2 +++++++++++++*)


	(*Valve 17, A+B*)
	(*spare*)
		Valve17FB
			(
			Enable_Motion:= Enable_Motion ,
			Enable_Latch:= TRUE,					(*Enabling Runs Valve as detent type (maintained solenoids*)
			Enable_SideA_PreCharge:= FALSE,		(*Enabling Turns Side A PreCharge Active, reset when Side B is energized in Auto*)
			Enable_SideB_PreCharge:= FALSE,		(*Enabling Turns Side B PreCharge Active, reset when Side A is energized in Auto*)
			PreCharge_Time:= T#0.1S,
			Enable_Auto_Commands:= In_Auto,
			Enable_Manual_Commands:= In_Manual AND All_Robots_Clear,
			In_Manual_SideA_Command:= Discrete_In.ManReqs2.0,
			In_Manual_SideB_Command:= (Discrete_In.ManReqs2.1 OR Discrete_In.Go_Home),
			SideA_Indicator:= FALSE,
			SideB_Indicator:= FALSE,
			TurnOn_SideA_SOL=> N101.Q.0,
			TurnOn_SideB_SOL=> N101.Q.1,
			TurnOn_SideA_Indicator=> Manual_Indicators2.0,
			TurnOn_SideB_Indicator=> Manual_Indicators2.1
			 );
		Valve17FB.In_Auto_SideA_Command:= FALSE;
		Valve17FB.In_Auto_SideB_Command:= FALSE;


	(*Valve 18, A+B*)
	(*spare*)
		Valve18FB
			(
			Enable_Motion:= Enable_Motion ,
			Enable_Latch:= TRUE,					(*Enabling Runs Valve as detent type (maintained solenoids*)
			Enable_SideA_PreCharge:= FALSE,		(*Enabling Turns Side A PreCharge Active, reset when Side B is energized in Auto*)
			Enable_SideB_PreCharge:= FALSE,		(*Enabling Turns Side B PreCharge Active, reset when Side A is energized in Auto*)
			PreCharge_Time:= T#0.10S,
			Enable_Auto_Commands:= In_Auto,
			Enable_Manual_Commands:= In_Manual AND All_Robots_Clear,
			In_Manual_SideA_Command:= Discrete_In.ManReqs2.2,
			In_Manual_SideB_Command:= Discrete_In.ManReqs2.3,
			SideA_Indicator:= FALSE,
			SideB_Indicator:= FALSE,
			TurnOn_SideA_SOL=> N101.Q.2,
			TurnOn_SideB_SOL=> N101.Q.3,
			TurnOn_SideA_Indicator=> Manual_Indicators2.2,
			TurnOn_SideB_Indicator=> Manual_Indicators2.3
			 );
		Valve18FB.In_Auto_SideA_Command:= FALSE;
		Valve18FB.In_Auto_SideB_Command:= FALSE;

	(*Valve 19, A+B*)
	(*spare*)
		Valve19FB
			(
			Enable_Motion:= Enable_Motion ,
			Enable_Latch:= TRUE,					(*Enabling Runs Valve as detent type (maintained solenoids*)
			Enable_SideA_PreCharge:= FALSE,		(*Enabling Turns Side A PreCharge Active, reset when Side B is energized in Auto*)
			Enable_SideB_PreCharge:= FALSE,		(*Enabling Turns Side B PreCharge Active, reset when Side A is energized in Auto*)
			PreCharge_Time:= T#0.10S,
			Enable_Auto_Commands:= In_Auto,
			Enable_Manual_Commands:= In_Manual AND All_Robots_Clear,
			In_Manual_SideA_Command:= Discrete_In.ManReqs2.4,
			In_Manual_SideB_Command:= Discrete_In.ManReqs2.5,
			SideA_Indicator:= FALSE,
			SideB_Indicator:= FALSE,
			TurnOn_SideA_SOL=> N101.Q.4,
			TurnOn_SideB_SOL=> N101.Q.5,
			TurnOn_SideA_Indicator=> Manual_Indicators2.4,
			TurnOn_SideB_Indicator=> Manual_Indicators2.5
			 );
		Valve19FB.In_Auto_SideA_Command:= FALSE;
		Valve19FB.In_Auto_SideB_Command:= FALSE;


	(*Valve 20, A+B*)
	(*spare*)
		Valve20FB
			(
			Enable_Motion:= Enable_Motion ,
			Enable_Latch:= TRUE,					(*Enabling Runs Valve as detent type (maintained solenoids*)
			Enable_SideA_PreCharge:= FALSE,		(*Enabling Turns Side A PreCharge Active, reset when Side B is energized in Auto*)
			Enable_SideB_PreCharge:= FALSE,		(*Enabling Turns Side B PreCharge Active, reset when Side A is energized in Auto*)
			PreCharge_Time:= T#0.10S,
			Enable_Auto_Commands:= In_Auto,
			Enable_Manual_Commands:= In_Manual AND All_Robots_Clear,
			In_Manual_SideA_Command:= Discrete_In.ManReqs2.6,
			In_Manual_SideB_Command:= Discrete_In.ManReqs2.7,
			SideA_Indicator:= FALSE,
			SideB_Indicator:= FALSE,
			TurnOn_SideA_SOL=> N101.Q.6,
			TurnOn_SideB_SOL=> N101.Q.7,
			TurnOn_SideA_Indicator=> Manual_Indicators2.6,
			TurnOn_SideB_Indicator=> Manual_Indicators2.7
			 );
		Valve20FB.In_Auto_SideA_Command:= FALSE;
		Valve20FB.In_Auto_SideB_Command:= FALSE;


	(*Valve 21, A+B*)
	(*spare*)
		Valve21FB
			(
			Enable_Motion:= Enable_Motion ,
			Enable_Latch:= TRUE,					(*Enabling Runs Valve as detent type (maintained solenoids*)
			Enable_SideA_PreCharge:= FALSE,		(*Enabling Turns Side A PreCharge Active, reset when Side B is energized in Auto*)
			Enable_SideB_PreCharge:= FALSE,		(*Enabling Turns Side B PreCharge Active, reset when Side A is energized in Auto*)
			PreCharge_Time:= T#0.10S,
			Enable_Auto_Commands:= In_Auto,
			Enable_Manual_Commands:= In_Manual AND All_Robots_Clear,
			In_Manual_SideA_Command:= Discrete_In.ManReqs2.8,
			In_Manual_SideB_Command:= Discrete_In.ManReqs2.9,
			SideA_Indicator:= FALSE,
			SideB_Indicator:= FALSE,
			TurnOn_SideA_SOL=> N101.Q.8,
			TurnOn_SideB_SOL=> N101.Q.9,
			TurnOn_SideA_Indicator=> Manual_Indicators2.8,
			TurnOn_SideB_Indicator=> Manual_Indicators2.9
			 );
		Valve21FB.In_Auto_SideA_Command:= FALSE;
		Valve21FB.In_Auto_SideB_Command:= FALSE;


	(*Valve 22, A+B*)
	(*spare*)
		Valve22FB
			(
			Enable_Motion:= Enable_Motion ,
			Enable_Latch:= TRUE,					(*Enabling Runs Valve as detent type (maintained solenoids*)
			Enable_SideA_PreCharge:= FALSE,		(*Enabling Turns Side A PreCharge Active, reset when Side B is energized in Auto*)
			Enable_SideB_PreCharge:= FALSE,		(*Enabling Turns Side B PreCharge Active, reset when Side A is energized in Auto*)
			PreCharge_Time:= T#0.10S,
			Enable_Auto_Commands:= In_Auto,
			Enable_Manual_Commands:= In_Manual AND All_Robots_Clear,
			In_Manual_SideA_Command:= Discrete_In.ManReqs2.10,
			In_Manual_SideB_Command:= Discrete_In.ManReqs2.11,
			SideA_Indicator:= FALSE,
			SideB_Indicator:= FALSE,
			TurnOn_SideA_SOL=> N101.Q.10,
			TurnOn_SideB_SOL=> N101.Q.11,
			TurnOn_SideA_Indicator=> Manual_Indicators2.10,
			TurnOn_SideB_Indicator=> Manual_Indicators2.11
			 );
		Valve22FB.In_Auto_SideA_Command:= FALSE;
		Valve22FB.In_Auto_SideB_Command:= FALSE;


	(*Valve 23, A+B*)
	(*spare*)
		Valve23FB
			(
			Enable_Motion:= Enable_Motion ,
			Enable_Latch:= TRUE,					(*Enabling Runs Valve as detent type (maintained solenoids*)
			Enable_SideA_PreCharge:= FALSE,		(*Enabling Turns Side A PreCharge Active, reset when Side B is energized in Auto*)
			Enable_SideB_PreCharge:= FALSE,		(*Enabling Turns Side B PreCharge Active, reset when Side A is energized in Auto*)
			PreCharge_Time:= T#0.10S,
			Enable_Auto_Commands:= In_Auto,
			Enable_Manual_Commands:= In_Manual AND All_Robots_Clear,
			In_Manual_SideA_Command:= Discrete_In.ManReqs2.12,
			In_Manual_SideB_Command:= Discrete_In.ManReqs2.13,
			SideA_Indicator:= FALSE,
			SideB_Indicator:= FALSE,
			TurnOn_SideA_SOL=> N101.Q.12,
			TurnOn_SideB_SOL=> N101.Q.13,
			TurnOn_SideA_Indicator=> Manual_Indicators2.12,
			TurnOn_SideB_Indicator=> Manual_Indicators2.13
			 );
		Valve23FB.In_Auto_SideA_Command:= FALSE;
		Valve23FB.In_Auto_SideB_Command:= FALSE;


	(*Valve 24, A+B*)
	(*spare*)
		Valve24FB
			(
			Enable_Motion:= Enable_Motion ,
			Enable_Latch:= TRUE,					(*Enabling Runs Valve as detent type (maintained solenoids*)
			Enable_SideA_PreCharge:= FALSE,		(*Enabling Turns Side A PreCharge Active, reset when Side B is energized in Auto*)
			Enable_SideB_PreCharge:= FALSE,		(*Enabling Turns Side B PreCharge Active, reset when Side A is energized in Auto*)
			PreCharge_Time:= T#0.10S,
			Enable_Auto_Commands:= In_Auto,
			Enable_Manual_Commands:= In_Manual AND All_Robots_Clear,
			In_Manual_SideA_Command:= Discrete_In.ManReqs2.14,
			In_Manual_SideB_Command:= Discrete_In.ManReqs2.15,
			SideA_Indicator:= FALSE,
			SideB_Indicator:= FALSE,
			TurnOn_SideA_SOL=> N101.Q.14,
			TurnOn_SideB_SOL=> N101.Q.15,
			TurnOn_SideA_Indicator=> Manual_Indicators2.14,
			TurnOn_SideB_Indicator=> Manual_Indicators2.15
			 );
		Valve24FB.In_Auto_SideA_Command:= FALSE;
		Valve24FB.In_Auto_SideB_Command:= FALSE;


	(*Valve 25, A+B*)
	(*spare*)
		Valve25FB
			(
			Enable_Motion:= Enable_Motion ,
			Enable_Latch:= TRUE,					(*Enabling Runs Valve as detent type (maintained solenoids*)
			Enable_SideA_PreCharge:= FALSE,		(*Enabling Turns Side A PreCharge Active, reset when Side B is energized in Auto*)
			Enable_SideB_PreCharge:= FALSE,		(*Enabling Turns Side B PreCharge Active, reset when Side A is energized in Auto*)
			PreCharge_Time:= T#0.10S,
			Enable_Auto_Commands:= In_Auto,
			Enable_Manual_Commands:= In_Manual AND All_Robots_Clear,
			In_Manual_SideA_Command:= Discrete_In.ManReqs2.16,
			In_Manual_SideB_Command:= Discrete_In.ManReqs2.17,
			SideA_Indicator:= FALSE,
			SideB_Indicator:= FALSE,
			TurnOn_SideA_SOL=> N101.Q.16,
			TurnOn_SideB_SOL=> N101.Q.17,
			TurnOn_SideA_Indicator=> Manual_Indicators2.16,
			TurnOn_SideB_Indicator=> Manual_Indicators2.17
			 );
		Valve25FB.In_Auto_SideA_Command:= FALSE;
		Valve25FB.In_Auto_SideB_Command:= FALSE;


	(*Valve 26, A+B*)
	(*spare*)
		Valve26FB
			(
			Enable_Motion:= Enable_Motion ,
			Enable_Latch:= TRUE,					(*Enabling Runs Valve as detent type (maintained solenoids*)
			Enable_SideA_PreCharge:= FALSE,		(*Enabling Turns Side A PreCharge Active, reset when Side B is energized in Auto*)
			Enable_SideB_PreCharge:= FALSE,		(*Enabling Turns Side B PreCharge Active, reset when Side A is energized in Auto*)
			PreCharge_Time:= T#0.10S,
			Enable_Auto_Commands:= In_Auto,
			Enable_Manual_Commands:= In_Manual AND All_Robots_Clear,
			In_Manual_SideA_Command:= Discrete_In.ManReqs2.18,
			In_Manual_SideB_Command:= Discrete_In.ManReqs2.19,
			SideA_Indicator:= FALSE,
			SideB_Indicator:= FALSE,
			TurnOn_SideA_SOL=> N101.Q.18,
			TurnOn_SideB_SOL=> N101.Q.19,
			TurnOn_SideA_Indicator=> Manual_Indicators2.18,
			TurnOn_SideB_Indicator=> Manual_Indicators2.19
			 );
		Valve26FB.In_Auto_SideA_Command:= FALSE;
		Valve26FB.In_Auto_SideB_Command:= FALSE;


	(*Valve 27, A+B*)
	(*spare*)
		Valve27FB
			(
			Enable_Motion:= Enable_Motion ,
			Enable_Latch:= TRUE,					(*Enabling Runs Valve as detent type (maintained solenoids*)
			Enable_SideA_PreCharge:= FALSE,		(*Enabling Turns Side A PreCharge Active, reset when Side B is energized in Auto*)
			Enable_SideB_PreCharge:= FALSE,		(*Enabling Turns Side B PreCharge Active, reset when Side A is energized in Auto*)
			PreCharge_Time:= T#0.10S,
			Enable_Auto_Commands:= In_Auto,
			Enable_Manual_Commands:= In_Manual AND All_Robots_Clear,
			In_Manual_SideA_Command:= Discrete_In.ManReqs2.20,
			In_Manual_SideB_Command:= Discrete_In.ManReqs2.21,
			SideA_Indicator:= FALSE,
			SideB_Indicator:= FALSE,
			TurnOn_SideA_SOL=> N101.Q.20,
			TurnOn_SideB_SOL=> N101.Q.21,
			TurnOn_SideA_Indicator=> Manual_Indicators2.20,
			TurnOn_SideB_Indicator=> Manual_Indicators2.21
			 );
		Valve27FB.In_Auto_SideA_Command:= FALSE;
		Valve27FB.In_Auto_SideB_Command:= FALSE;


	(*Valve 28, A+B*)
	(*spare*)
		Valve28FB
			(
			Enable_Motion:= Enable_Motion ,
			Enable_Latch:= TRUE,					(*Enabling Runs Valve as detent type (maintained solenoids*)
			Enable_SideA_PreCharge:= FALSE,		(*Enabling Turns Side A PreCharge Active, reset when Side B is energized in Auto*)
			Enable_SideB_PreCharge:= FALSE,		(*Enabling Turns Side B PreCharge Active, reset when Side A is energized in Auto*)
			PreCharge_Time:= T#0.10S,
			Enable_Auto_Commands:= In_Auto,
			Enable_Manual_Commands:= In_Manual AND All_Robots_Clear,
			In_Manual_SideA_Command:= Discrete_In.ManReqs2.22,
			In_Manual_SideB_Command:= Discrete_In.ManReqs2.23,
			SideA_Indicator:= FALSE,
			SideB_Indicator:= FALSE,
			TurnOn_SideA_SOL=> N101.Q.22,
			TurnOn_SideB_SOL=> N101.Q.23,
			TurnOn_SideA_Indicator=> Manual_Indicators2.22,
			TurnOn_SideB_Indicator=> Manual_Indicators2.23
			 );
		Valve28FB.In_Auto_SideA_Command:= FALSE;
		Valve28FB.In_Auto_SideB_Command:= FALSE;


	(*Valve 29, A+B*)
	(*spare*)
		Valve29FB
			(
			Enable_Motion:= Enable_Motion ,
			Enable_Latch:= TRUE,					(*Enabling Runs Valve as detent type (maintained solenoids*)
			Enable_SideA_PreCharge:= FALSE,		(*Enabling Turns Side A PreCharge Active, reset when Side B is energized in Auto*)
			Enable_SideB_PreCharge:= FALSE,		(*Enabling Turns Side B PreCharge Active, reset when Side A is energized in Auto*)
			PreCharge_Time:= T#0.10S,
			Enable_Auto_Commands:= In_Auto,
			Enable_Manual_Commands:= In_Manual AND All_Robots_Clear,
			In_Manual_SideA_Command:= Discrete_In.ManReqs2.24,
			In_Manual_SideB_Command:= Discrete_In.ManReqs2.25,
			SideA_Indicator:= FALSE,
			SideB_Indicator:= FALSE,
			TurnOn_SideA_SOL=> N101.Q.24,
			TurnOn_SideB_SOL=> N101.Q.25,
			TurnOn_SideA_Indicator=> Manual_Indicators2.24,
			TurnOn_SideB_Indicator=> Manual_Indicators2.25
			 );
		Valve29FB.In_Auto_SideA_Command:= FALSE;
		Valve29FB.In_Auto_SideB_Command:= FALSE;


	(*Valve 30, A+B*)
	(*spare*)
		Valve30FB
			(
			Enable_Motion:= Enable_Motion ,
			Enable_Latch:= TRUE,					(*Enabling Runs Valve as detent type (maintained solenoids*)
			Enable_SideA_PreCharge:= FALSE,		(*Enabling Turns Side A PreCharge Active, reset when Side B is energized in Auto*)
			Enable_SideB_PreCharge:= FALSE,		(*Enabling Turns Side B PreCharge Active, reset when Side A is energized in Auto*)
			PreCharge_Time:= T#0.10S,
			Enable_Auto_Commands:= In_Auto,
			Enable_Manual_Commands:= In_Manual AND All_Robots_Clear,
			In_Manual_SideA_Command:= Discrete_In.ManReqs2.26,
			In_Manual_SideB_Command:= Discrete_In.ManReqs2.27,
			SideA_Indicator:= FALSE,
			SideB_Indicator:= FALSE,
			TurnOn_SideA_SOL=> N101.Q.26,
			TurnOn_SideB_SOL=> N101.Q.27,
			TurnOn_SideA_Indicator=> Manual_Indicators2.26,
			TurnOn_SideB_Indicator=> Manual_Indicators2.27
			 );
		Valve30FB.In_Auto_SideA_Command:= FALSE;
		Valve30FB.In_Auto_SideB_Command:= FALSE;


	(*Valve 31, A+B*)
	(*spare*)
		Valve31FB
			(
			Enable_Motion:= Enable_Motion ,
			Enable_Latch:= TRUE,					(*Enabling Runs Valve as detent type (maintained solenoids*)
			Enable_SideA_PreCharge:= FALSE,		(*Enabling Turns Side A PreCharge Active, reset when Side B is energized in Auto*)
			Enable_SideB_PreCharge:= FALSE,		(*Enabling Turns Side B PreCharge Active, reset when Side A is energized in Auto*)
			PreCharge_Time:= T#0.10S,
			Enable_Auto_Commands:= In_Auto,
			Enable_Manual_Commands:= In_Manual AND All_Robots_Clear,
			In_Manual_SideA_Command:= Discrete_In.ManReqs2.28,
			In_Manual_SideB_Command:= Discrete_In.ManReqs2.29,
			SideA_Indicator:= FALSE,
			SideB_Indicator:= FALSE,
			TurnOn_SideA_SOL=> N101.Q.28,
			TurnOn_SideB_SOL=> N101.Q.29,
			TurnOn_SideA_Indicator=> Manual_Indicators2.28,
			TurnOn_SideB_Indicator=> Manual_Indicators2.29
			 );
		Valve31FB.In_Auto_SideA_Command:= FALSE;
		Valve31FB.In_Auto_SideB_Command:= FALSE;


	(*Valve 32, A+B*)
	(*spare*)
		Valve32FB
			(
			Enable_Motion:= Enable_Motion ,
			Enable_Latch:= TRUE,					(*Enabling Runs Valve as detent type (maintained solenoids*)
			Enable_SideA_PreCharge:= FALSE,		(*Enabling Turns Side A PreCharge Active, reset when Side B is energized in Auto*)
			Enable_SideB_PreCharge:= FALSE,		(*Enabling Turns Side B PreCharge Active, reset when Side A is energized in Auto*)
			PreCharge_Time:= T#0.10S,
			Enable_Auto_Commands:= In_Auto,
			Enable_Manual_Commands:= In_Manual AND All_Robots_Clear,
			In_Manual_SideA_Command:= Discrete_In.ManReqs2.30,
			In_Manual_SideB_Command:= Discrete_In.ManReqs2.31,
			SideA_Indicator:= FALSE,
			SideB_Indicator:= FALSE,
			TurnOn_SideA_SOL=> N101.Q.30,
			TurnOn_SideB_SOL=> N101.Q.31,
			TurnOn_SideA_Indicator=> Manual_Indicators2.30,
			TurnOn_SideB_Indicator=> Manual_Indicators2.31
			 );
		Valve32FB.In_Auto_SideA_Command:= FALSE;
		Valve32FB.In_Auto_SideB_Command:= FALSE;




















(*end*)
END_ACTION

ACTION ValveBank3:


(*+++++++++++THIS AREA IS CUSTOM PER INSTALLATION AND WILL HAVE TO BE MODIFIED PER +++++++++++++*)
(*+++++++++++THIS AREA IS CUSTOM PER INSTALLATION AND WILL HAVE TO BE MODIFIED PER +++++++++++++*)
(*+++++++++++THIS AREA IS CUSTOM PER INSTALLATION AND WILL HAVE TO BE MODIFIED PER +++++++++++++*)

(*+++++++++++VALVE BANK 3 +++++++++++++*)
(*+++++++++++VALVE BANK 3 +++++++++++++*)
(*+++++++++++VALVE BANK 3 +++++++++++++*)


	(*Valve 33, A+B*)
	(*spare*)
		Valve33FB
			(
			Enable_Motion:= Enable_Motion ,
			Enable_Latch:= TRUE,					(*Enabling Runs Valve as detent type (maintained solenoids*)
			Enable_SideA_PreCharge:= FALSE,		(*Enabling Turns Side A PreCharge Active, reset when Side B is energized in Auto*)
			Enable_SideB_PreCharge:= FALSE,		(*Enabling Turns Side B PreCharge Active, reset when Side A is energized in Auto*)
			PreCharge_Time:= T#0.1S,
			Enable_Auto_Commands:= In_Auto,
			Enable_Manual_Commands:= In_Manual AND All_Robots_Clear,
			In_Manual_SideA_Command:= Discrete_In.ManReqs3.0,
			In_Manual_SideB_Command:= (Discrete_In.ManReqs3.1 OR Discrete_In.Go_Home),
			SideA_Indicator:= FALSE,
			SideB_Indicator:= FALSE,
			TurnOn_SideA_SOL=> N102.Q.0,
			TurnOn_SideB_SOL=> N102.Q.1,
			TurnOn_SideA_Indicator=> Manual_Indicators3.0,
			TurnOn_SideB_Indicator=> Manual_Indicators3.1
			 );
		Valve33FB.In_Auto_SideA_Command:= FALSE;
		Valve33FB.In_Auto_SideB_Command:= FALSE;


	(*Valve 34, A+B*)
	(*spare*)
		Valve34FB
			(
			Enable_Motion:= Enable_Motion ,
			Enable_Latch:= TRUE,					(*Enabling Runs Valve as detent type (maintained solenoids*)
			Enable_SideA_PreCharge:= FALSE,		(*Enabling Turns Side A PreCharge Active, reset when Side B is energized in Auto*)
			Enable_SideB_PreCharge:= FALSE,		(*Enabling Turns Side B PreCharge Active, reset when Side A is energized in Auto*)
			PreCharge_Time:= T#0.10S,
			Enable_Auto_Commands:= In_Auto,
			Enable_Manual_Commands:= In_Manual AND All_Robots_Clear,
			In_Manual_SideA_Command:= Discrete_In.ManReqs3.2,
			In_Manual_SideB_Command:= Discrete_In.ManReqs3.3,
			SideA_Indicator:= FALSE,
			SideB_Indicator:= FALSE,
			TurnOn_SideA_SOL=> N102.Q.2,
			TurnOn_SideB_SOL=> N102.Q.3,
			TurnOn_SideA_Indicator=> Manual_Indicators3.2,
			TurnOn_SideB_Indicator=> Manual_Indicators3.3
			 );
		Valve34FB.In_Auto_SideA_Command:= FALSE;
		Valve34FB.In_Auto_SideB_Command:= FALSE;


	(*Valve 35, A+B*)
	(*spare*)
		Valve35FB
			(
			Enable_Motion:= Enable_Motion ,
			Enable_Latch:= TRUE,					(*Enabling Runs Valve as detent type (maintained solenoids*)
			Enable_SideA_PreCharge:= FALSE,		(*Enabling Turns Side A PreCharge Active, reset when Side B is energized in Auto*)
			Enable_SideB_PreCharge:= FALSE,		(*Enabling Turns Side B PreCharge Active, reset when Side A is energized in Auto*)
			PreCharge_Time:= T#0.10S,
			Enable_Auto_Commands:= In_Auto,
			Enable_Manual_Commands:= In_Manual AND All_Robots_Clear,
			In_Manual_SideA_Command:= Discrete_In.ManReqs3.4,
			In_Manual_SideB_Command:= Discrete_In.ManReqs3.5,
			SideA_Indicator:= FALSE,
			SideB_Indicator:= FALSE,
			TurnOn_SideA_SOL=> N102.Q.4,
			TurnOn_SideB_SOL=> N102.Q.5,
			TurnOn_SideA_Indicator=> Manual_Indicators3.4,
			TurnOn_SideB_Indicator=> Manual_Indicators3.5
			 );
		Valve35FB.In_Auto_SideA_Command:= FALSE;
		Valve35FB.In_Auto_SideB_Command:= FALSE;


	(*Valve 36, A+B*)
	(*spare*)
		Valve36FB
			(
			Enable_Motion:= Enable_Motion ,
			Enable_Latch:= TRUE,					(*Enabling Runs Valve as detent type (maintained solenoids*)
			Enable_SideA_PreCharge:= FALSE,		(*Enabling Turns Side A PreCharge Active, reset when Side B is energized in Auto*)
			Enable_SideB_PreCharge:= FALSE,		(*Enabling Turns Side B PreCharge Active, reset when Side A is energized in Auto*)
			PreCharge_Time:= T#0.10S,
			Enable_Auto_Commands:= In_Auto,
			Enable_Manual_Commands:= In_Manual AND All_Robots_Clear,
			In_Manual_SideA_Command:= Discrete_In.ManReqs3.6,
			In_Manual_SideB_Command:= Discrete_In.ManReqs3.7,
			SideA_Indicator:= FALSE,
			SideB_Indicator:= FALSE,
			TurnOn_SideA_SOL=> N102.Q.6,
			TurnOn_SideB_SOL=> N102.Q.7,
			TurnOn_SideA_Indicator=> Manual_Indicators3.6,
			TurnOn_SideB_Indicator=> Manual_Indicators3.7
			 );
		Valve36FB.In_Auto_SideA_Command:= FALSE;
		Valve36FB.In_Auto_SideB_Command:= FALSE;


	(*Valve 37, A+B*)
	(*spare*)
		Valve37FB
			(
			Enable_Motion:= Enable_Motion ,
			Enable_Latch:= TRUE,					(*Enabling Runs Valve as detent type (maintained solenoids*)
			Enable_SideA_PreCharge:= FALSE,		(*Enabling Turns Side A PreCharge Active, reset when Side B is energized in Auto*)
			Enable_SideB_PreCharge:= FALSE,		(*Enabling Turns Side B PreCharge Active, reset when Side A is energized in Auto*)
			PreCharge_Time:= T#0.10S,
			Enable_Auto_Commands:= In_Auto,
			Enable_Manual_Commands:= In_Manual AND All_Robots_Clear,
			In_Manual_SideA_Command:= Discrete_In.ManReqs3.8,
			In_Manual_SideB_Command:= Discrete_In.ManReqs3.9,
			SideA_Indicator:= FALSE,
			SideB_Indicator:= FALSE,
			TurnOn_SideA_SOL=> N102.Q.8,
			TurnOn_SideB_SOL=> N102.Q.9,
			TurnOn_SideA_Indicator=> Manual_Indicators3.8,
			TurnOn_SideB_Indicator=> Manual_Indicators3.9
			 );
		Valve37FB.In_Auto_SideA_Command:= FALSE;
		Valve37FB.In_Auto_SideB_Command:= FALSE;


	(*Valve 38, A+B*)
	(*spare*)
		Valve38FB
			(
			Enable_Motion:= Enable_Motion ,
			Enable_Latch:= TRUE,					(*Enabling Runs Valve as detent type (maintained solenoids*)
			Enable_SideA_PreCharge:= FALSE,		(*Enabling Turns Side A PreCharge Active, reset when Side B is energized in Auto*)
			Enable_SideB_PreCharge:= FALSE,		(*Enabling Turns Side B PreCharge Active, reset when Side A is energized in Auto*)
			PreCharge_Time:= T#0.10S,
			Enable_Auto_Commands:= In_Auto,
			Enable_Manual_Commands:= In_Manual AND All_Robots_Clear,
			In_Manual_SideA_Command:= Discrete_In.ManReqs3.10,
			In_Manual_SideB_Command:= Discrete_In.ManReqs3.11,
			SideA_Indicator:= FALSE,
			SideB_Indicator:= FALSE,
			TurnOn_SideA_SOL=> N102.Q.10,
			TurnOn_SideB_SOL=> N102.Q.11,
			TurnOn_SideA_Indicator=> Manual_Indicators3.10,
			TurnOn_SideB_Indicator=> Manual_Indicators3.11
			 );
		Valve38FB.In_Auto_SideA_Command:= FALSE;
		Valve38FB.In_Auto_SideB_Command:= FALSE;


	(*Valve 39, A+B*)
	(*spare*)
		Valve39FB
			(
			Enable_Motion:= Enable_Motion ,
			Enable_Latch:= TRUE,					(*Enabling Runs Valve as detent type (maintained solenoids*)
			Enable_SideA_PreCharge:= FALSE,		(*Enabling Turns Side A PreCharge Active, reset when Side B is energized in Auto*)
			Enable_SideB_PreCharge:= FALSE,		(*Enabling Turns Side B PreCharge Active, reset when Side A is energized in Auto*)
			PreCharge_Time:= T#0.10S,
			Enable_Auto_Commands:= In_Auto,
			Enable_Manual_Commands:= In_Manual AND All_Robots_Clear,
			In_Manual_SideA_Command:= Discrete_In.ManReqs3.12,
			In_Manual_SideB_Command:= Discrete_In.ManReqs3.13,
			SideA_Indicator:= FALSE,
			SideB_Indicator:= FALSE,
			TurnOn_SideA_SOL=> N102.Q.12,
			TurnOn_SideB_SOL=> N102.Q.13,
			TurnOn_SideA_Indicator=> Manual_Indicators3.12,
			TurnOn_SideB_Indicator=> Manual_Indicators3.13
			 );
		Valve39FB.In_Auto_SideA_Command:= FALSE;
		Valve39FB.In_Auto_SideB_Command:= FALSE;


	(*Valve 40, A+B*)
	(*spare*)
		Valve40FB
			(
			Enable_Motion:= Enable_Motion ,
			Enable_Latch:= TRUE,					(*Enabling Runs Valve as detent type (maintained solenoids*)
			Enable_SideA_PreCharge:= FALSE,		(*Enabling Turns Side A PreCharge Active, reset when Side B is energized in Auto*)
			Enable_SideB_PreCharge:= FALSE,		(*Enabling Turns Side B PreCharge Active, reset when Side A is energized in Auto*)
			PreCharge_Time:= T#0.10S,
			Enable_Auto_Commands:= In_Auto,
			Enable_Manual_Commands:= In_Manual AND All_Robots_Clear,
			In_Manual_SideA_Command:= Discrete_In.ManReqs3.14,
			In_Manual_SideB_Command:= Discrete_In.ManReqs3.15,
			SideA_Indicator:= FALSE,
			SideB_Indicator:= FALSE,
			TurnOn_SideA_SOL=> N102.Q.14,
			TurnOn_SideB_SOL=> N102.Q.15,
			TurnOn_SideA_Indicator=> Manual_Indicators3.14,
			TurnOn_SideB_Indicator=> Manual_Indicators3.15
			 );
		Valve40FB.In_Auto_SideA_Command:= FALSE;
		Valve40FB.In_Auto_SideB_Command:= FALSE;


	(*Valve 41, A+B*)
	(*spare*)
		Valve41FB
			(
			Enable_Motion:= Enable_Motion ,
			Enable_Latch:= TRUE,					(*Enabling Runs Valve as detent type (maintained solenoids*)
			Enable_SideA_PreCharge:= FALSE,		(*Enabling Turns Side A PreCharge Active, reset when Side B is energized in Auto*)
			Enable_SideB_PreCharge:= FALSE,		(*Enabling Turns Side B PreCharge Active, reset when Side A is energized in Auto*)
			PreCharge_Time:= T#0.10S,
			Enable_Auto_Commands:= In_Auto,
			Enable_Manual_Commands:= In_Manual AND All_Robots_Clear,
			In_Manual_SideA_Command:= Discrete_In.ManReqs3.16,
			In_Manual_SideB_Command:= Discrete_In.ManReqs3.17,
			SideA_Indicator:= FALSE,
			SideB_Indicator:= FALSE,
			TurnOn_SideA_SOL=> N102.Q.16,
			TurnOn_SideB_SOL=> N102.Q.17,
			TurnOn_SideA_Indicator=> Manual_Indicators3.16,
			TurnOn_SideB_Indicator=> Manual_Indicators3.17
			 );
		Valve41FB.In_Auto_SideA_Command:= FALSE;
		Valve41FB.In_Auto_SideB_Command:= FALSE;


	(*Valve 42, A+B*)
	(*spare*)
		Valve42FB
			(
			Enable_Motion:= Enable_Motion ,
			Enable_Latch:= TRUE,					(*Enabling Runs Valve as detent type (maintained solenoids*)
			Enable_SideA_PreCharge:= FALSE,		(*Enabling Turns Side A PreCharge Active, reset when Side B is energized in Auto*)
			Enable_SideB_PreCharge:= FALSE,		(*Enabling Turns Side B PreCharge Active, reset when Side A is energized in Auto*)
			PreCharge_Time:= T#0.10S,
			Enable_Auto_Commands:= In_Auto,
			Enable_Manual_Commands:= In_Manual AND All_Robots_Clear,
			In_Manual_SideA_Command:= Discrete_In.ManReqs3.18,
			In_Manual_SideB_Command:= Discrete_In.ManReqs3.19,
			SideA_Indicator:= FALSE,
			SideB_Indicator:= FALSE,
			TurnOn_SideA_SOL=> N102.Q.18,
			TurnOn_SideB_SOL=> N102.Q.19,
			TurnOn_SideA_Indicator=> Manual_Indicators3.18,
			TurnOn_SideB_Indicator=> Manual_Indicators3.19
			 );
		Valve42FB.In_Auto_SideA_Command:= FALSE;
		Valve42FB.In_Auto_SideB_Command:= FALSE;


	(*Valve 43, A+B*)
	(*spare*)
		Valve43FB
			(
			Enable_Motion:= Enable_Motion ,
			Enable_Latch:= TRUE,					(*Enabling Runs Valve as detent type (maintained solenoids*)
			Enable_SideA_PreCharge:= FALSE,		(*Enabling Turns Side A PreCharge Active, reset when Side B is energized in Auto*)
			Enable_SideB_PreCharge:= FALSE,		(*Enabling Turns Side B PreCharge Active, reset when Side A is energized in Auto*)
			PreCharge_Time:= T#0.10S,
			Enable_Auto_Commands:= In_Auto,
			Enable_Manual_Commands:= In_Manual AND All_Robots_Clear,
			In_Manual_SideA_Command:= Discrete_In.ManReqs3.20,
			In_Manual_SideB_Command:= Discrete_In.ManReqs3.21,
			SideA_Indicator:= FALSE,
			SideB_Indicator:= FALSE,
			TurnOn_SideA_SOL=> N102.Q.20,
			TurnOn_SideB_SOL=> N102.Q.21,
			TurnOn_SideA_Indicator=> Manual_Indicators3.20,
			TurnOn_SideB_Indicator=> Manual_Indicators3.21
			 );
		Valve43FB.In_Auto_SideA_Command:= FALSE;
		Valve43FB.In_Auto_SideB_Command:= FALSE;


	(*Valve 44, A+B*)
	(*spare*)
		Valve44FB
			(
			Enable_Motion:= Enable_Motion ,
			Enable_Latch:= TRUE,					(*Enabling Runs Valve as detent type (maintained solenoids*)
			Enable_SideA_PreCharge:= FALSE,		(*Enabling Turns Side A PreCharge Active, reset when Side B is energized in Auto*)
			Enable_SideB_PreCharge:= FALSE,		(*Enabling Turns Side B PreCharge Active, reset when Side A is energized in Auto*)
			PreCharge_Time:= T#0.10S,
			Enable_Auto_Commands:= In_Auto,
			Enable_Manual_Commands:= In_Manual AND All_Robots_Clear,
			In_Manual_SideA_Command:= Discrete_In.ManReqs3.22,
			In_Manual_SideB_Command:= Discrete_In.ManReqs3.23,
			SideA_Indicator:= FALSE,
			SideB_Indicator:= FALSE,
			TurnOn_SideA_SOL=> N102.Q.22,
			TurnOn_SideB_SOL=> N102.Q.23,
			TurnOn_SideA_Indicator=> Manual_Indicators3.22,
			TurnOn_SideB_Indicator=> Manual_Indicators3.23
			 );
		Valve44FB.In_Auto_SideA_Command:= FALSE;
		Valve44FB.In_Auto_SideB_Command:= FALSE;


	(*Valve 45, A+B*)
	(*spare*)
		Valve45FB
			(
			Enable_Motion:= Enable_Motion ,
			Enable_Latch:= TRUE,					(*Enabling Runs Valve as detent type (maintained solenoids*)
			Enable_SideA_PreCharge:= FALSE,		(*Enabling Turns Side A PreCharge Active, reset when Side B is energized in Auto*)
			Enable_SideB_PreCharge:= FALSE,		(*Enabling Turns Side B PreCharge Active, reset when Side A is energized in Auto*)
			PreCharge_Time:= T#0.10S,
			Enable_Auto_Commands:= In_Auto,
			Enable_Manual_Commands:= In_Manual AND All_Robots_Clear,
			In_Manual_SideA_Command:= Discrete_In.ManReqs3.24,
			In_Manual_SideB_Command:= Discrete_In.ManReqs3.25,
			SideA_Indicator:= FALSE,
			SideB_Indicator:= FALSE,
			TurnOn_SideA_SOL=> N102.Q.24,
			TurnOn_SideB_SOL=> N102.Q.25,
			TurnOn_SideA_Indicator=> Manual_Indicators3.24,
			TurnOn_SideB_Indicator=> Manual_Indicators3.25
			 );
		Valve45FB.In_Auto_SideA_Command:= FALSE;
		Valve45FB.In_Auto_SideB_Command:= FALSE;


	(*Valve 46, A+B*)
	(*spare*)
		Valve46FB
			(
			Enable_Motion:= Enable_Motion ,
			Enable_Latch:= TRUE,					(*Enabling Runs Valve as detent type (maintained solenoids*)
			Enable_SideA_PreCharge:= FALSE,		(*Enabling Turns Side A PreCharge Active, reset when Side B is energized in Auto*)
			Enable_SideB_PreCharge:= FALSE,		(*Enabling Turns Side B PreCharge Active, reset when Side A is energized in Auto*)
			PreCharge_Time:= T#0.10S,
			Enable_Auto_Commands:= In_Auto,
			Enable_Manual_Commands:= In_Manual AND All_Robots_Clear,
			In_Manual_SideA_Command:= Discrete_In.ManReqs3.26,
			In_Manual_SideB_Command:= Discrete_In.ManReqs3.27,
			SideA_Indicator:= FALSE,
			SideB_Indicator:= FALSE,
			TurnOn_SideA_SOL=> N102.Q.26,
			TurnOn_SideB_SOL=> N102.Q.27,
			TurnOn_SideA_Indicator=> Manual_Indicators3.26,
			TurnOn_SideB_Indicator=> Manual_Indicators3.27
			 );
		Valve46FB.In_Auto_SideA_Command:= FALSE;
		Valve46FB.In_Auto_SideB_Command:= FALSE;


	(*Valve 47, A+B*)
	(*spare*)
		Valve47FB
			(
			Enable_Motion:= Enable_Motion ,
			Enable_Latch:= TRUE,					(*Enabling Runs Valve as detent type (maintained solenoids*)
			Enable_SideA_PreCharge:= FALSE,		(*Enabling Turns Side A PreCharge Active, reset when Side B is energized in Auto*)
			Enable_SideB_PreCharge:= FALSE,		(*Enabling Turns Side B PreCharge Active, reset when Side A is energized in Auto*)
			PreCharge_Time:= T#0.10S,
			Enable_Auto_Commands:= In_Auto,
			Enable_Manual_Commands:= In_Manual AND All_Robots_Clear,
			In_Manual_SideA_Command:= Discrete_In.ManReqs3.28,
			In_Manual_SideB_Command:= Discrete_In.ManReqs3.29,
			SideA_Indicator:= FALSE,
			SideB_Indicator:= FALSE,
			TurnOn_SideA_SOL=> N102.Q.28,
			TurnOn_SideB_SOL=> N102.Q.29,
			TurnOn_SideA_Indicator=> Manual_Indicators3.28,
			TurnOn_SideB_Indicator=> Manual_Indicators3.29
			 );
		Valve47FB.In_Auto_SideA_Command:= FALSE;
		Valve47FB.In_Auto_SideB_Command:= FALSE;


	(*Valve 48, A+B*)
	(*spare*)
		Valve48FB
			(
			Enable_Motion:= Enable_Motion ,
			Enable_Latch:= TRUE,					(*Enabling Runs Valve as detent type (maintained solenoids*)
			Enable_SideA_PreCharge:= FALSE,		(*Enabling Turns Side A PreCharge Active, reset when Side B is energized in Auto*)
			Enable_SideB_PreCharge:= FALSE,		(*Enabling Turns Side B PreCharge Active, reset when Side A is energized in Auto*)
			PreCharge_Time:= T#0.10S,
			Enable_Auto_Commands:= In_Auto,
			Enable_Manual_Commands:= In_Manual AND All_Robots_Clear,
			In_Manual_SideA_Command:= Discrete_In.ManReqs3.30,
			In_Manual_SideB_Command:= Discrete_In.ManReqs3.31,
			SideA_Indicator:= FALSE,
			SideB_Indicator:= FALSE,
			TurnOn_SideA_SOL=> N102.Q.30,
			TurnOn_SideB_SOL=> N102.Q.31,
			TurnOn_SideA_Indicator=> Manual_Indicators3.30,
			TurnOn_SideB_Indicator=> Manual_Indicators3.31
			 );
		Valve48FB.In_Auto_SideA_Command:= FALSE;
		Valve48FB.In_Auto_SideB_Command:= FALSE;


























(*end*)
END_ACTION

ACTION Xfer_To_UI:
(*Transfer General Status of Fixture and I/O Images for Display On HMI*)
	Discrete_Image.Status:= Status;
	Discrete_Image.CLFaults1:= CLFaults1;
	Discrete_Image.CLFaults2:= CLFaults2;
	Discrete_Image.CLFaults3:= CLFaults3;
	Discrete_Image.CLFaults4:= CLFaults4;
	Discrete_Image.CLFaulted:= CLFaulted;
	Discrete_Image.PPFaults:= PPFaults;
	Discrete_Image.PPFaults1:= PPFaults1;
	Discrete_Image.PPFaults2:= PPFaults2;
	Discrete_Image.PPFaulted:= PPFaulted;
	Discrete_Image.Model_Data:= Model_ID;
	Discrete_Image.ToolID:= Fix_ID;
	Discrete_Image.ProdCount:= Prod_Count_Out;
	Discrete_Image.CycleTime:= Cycle_Time_Out;
	Discrete_Image.PrevCycleTime:= PrevCycle_Time_Out;
	Discrete_Image.LoadTime:= Load_Time_Out;
	Discrete_Image.WeldTime:= Weld_Time_Out;
	Discrete_Image.UnloadTime:= Unload_Time_Out;

	Discrete_Image.InAuto:= In_Auto_Mode;
	Discrete_Image.InManual:= In_Manual_Mode;
	Discrete_Image.ManInds:= Manual_Indicators1;
	Discrete_Image.ManInds2:= Manual_Indicators2;
	Discrete_Image.ManInds3:= Manual_Indicators3;
	Discrete_Image.At_Home:= Tool_At_Home;
	Discrete_Image.Enable_Motion:= Enable_Motion;
	Discrete_Image.All_Sensors_Off:= All_Sensors_Off;
	Discrete_Image.Bypass_ACKS:= Discrete_In.Bypass_REQS;
	Discrete_Image.CustomApplication_ACKS:= Discrete_In.CustomApplication_REQS;
	Discrete_Image.Fixture_Allow_Model_Change:= Fixture_Allow_Model_Change;
	Discrete_Image.NodeLayout:=NodeLayout;
	Discrete_Image.NodeState:=NodeState;
	
	Discrete_Image.Input_Node_Count:= Discrete_In.Input_Node_Count;
	Discrete_Image.VB_Node_Count:= Discrete_In.VB_Node_Count;
	Discrete_Image.Water_Stand_Count:= Discrete_In.Water_Stand_Count;

	IF  (Discrete_Image.Input_Node_Count < 4)
		THEN Discrete_Image.VB_Screen_Position:= 1;
	ELSIF  (Discrete_Image.Input_Node_Count < 7)
		THEN Discrete_Image.VB_Screen_Position:= 2;
	ELSIF  (Discrete_Image.Input_Node_Count < 10)
		THEN Discrete_Image.VB_Screen_Position:= 3;
	ELSIF  (Discrete_Image.Input_Node_Count < 13)
		THEN Discrete_Image.VB_Screen_Position:= 4;
	ELSIF  (Discrete_Image.Input_Node_Count < 16)
		THEN Discrete_Image.VB_Screen_Position:= 5;
	ELSIF  (Discrete_Image.Input_Node_Count < 19)
		THEN Discrete_Image.VB_Screen_Position:= 6;
	ELSIF  (Discrete_Image.Input_Node_Count < 22)
		THEN Discrete_Image.VB_Screen_Position:= 7;
	ELSIF  (Discrete_Image.Input_Node_Count < 26)
		THEN Discrete_Image.VB_Screen_Position:= 8;
	ELSE
			Discrete_Image.VB_Screen_Position:= 9;
	END_IF;

	Discrete_Image.N00:= N00;
	Discrete_Image.N01:= N01;
	Discrete_Image.N02:= N02;
	Discrete_Image.N03:= N03;
	Discrete_Image.N04:= N04;
	Discrete_Image.N05:= N05;
	Discrete_Image.N06:= N06;
	Discrete_Image.N07:= N07;
	Discrete_Image.N08:= N08;
	Discrete_Image.N09:= N09;
	Discrete_Image.N10:= N10;
	Discrete_Image.N11:= N11;
	Discrete_Image.N12:= N12;
	Discrete_Image.N13:= N13;
	Discrete_Image.N14:= N14;
	Discrete_Image.N15:= N15;
	Discrete_Image.N16:= N16;
	Discrete_Image.N17:= N17;
	Discrete_Image.N18:= N18;
	Discrete_Image.N19:= N19;
	Discrete_Image.N100:= N100;
	Discrete_Image.N100_STAT:= N100_STAT;
	Discrete_Image.N101:= N101;
	Discrete_Image.N101_STAT:= N101_STAT;
	Discrete_Image.N102:= N102;
	Discrete_Image.N102_STAT:= N102_STAT;


	Discrete_Image.ECatSlave_Cable_Breaks:= ECatSlave_Cable_Breaks;

	Discrete_Image.Operator_Performance_Pen:= Production_Report.Shift_Report[0].Prod_Performance;
END_ACTION

END_PROGRAM

(* stored: Version 1.1.0.1, ProductVersion 3.1.4024.12
   POU Fix112: Id {d420705a-7532-4fd0-abd8-d2a998a318ed}, SpecialFunc None
   Action All_Sensors: Id {b40a21dd-55b5-4194-ac23-b384f1e308b5}
   Action Cylinders: Id {2b45d9ee-6836-4de4-9d44-ab93a19fd01e}
   Action Hardware: Id {9ab411df-27f3-4a28-adeb-58ff5886e9fe}
   Action Production: Id {de59f99a-122c-4124-83ab-fd0fb99d4c53}
   Action Proxies: Id {8f4157f0-da54-4e34-b4c0-16054aa889f7}
   Action Robot_Registration: Id {d1ecc0fc-751e-43ea-826f-4c8d8f447aa8}
   Action Status_and_Faults: Id {f16b3ae2-d157-40d9-8ada-f19b173bfa05}
   Action Task_Fix_Model_IDs: Id {4914d2c8-3872-46a1-b6a4-56edf1efb7bb}
   Action Tool_States: Id {86aadd8b-44f9-4a0c-84e7-3414feea4032}
   Action Tool_VBSeq_Repos: Id {cb5d67ef-173e-4012-90bc-764c15190993}
   Action ValveBank1: Id {7b46ebfe-7d29-45fc-9d7b-d9d73250f840}
   Action ValveBank2: Id {a3c5d8cd-2e7e-421d-b730-226142413706}
   Action ValveBank3: Id {0eb00167-b347-42e8-837a-871fe935163a}
   Action Xfer_To_UI: Id {daf228c6-fbe2-4234-bea4-9106f9042f7c} *)
